FUNCTION_BLOCK MECH2_MDL (* Motion/Fault Model of a Bidirectional Linear Mechanism (Externally Clocked) *)
  (* Standard: 61499-1; Classification: Model; ApplicationDomain: Simulation; Function: Bidirectional Motion *)
  (* Version 0.0, 2004-09-25, JHC, Rockwell Automation, Derived from MECH2_MDL. *)
  (* Compiler header: package fb.rt.mva; import fb.rt.math.*; *)
  (* Compiler Java IBM Jikes 1.06 *)
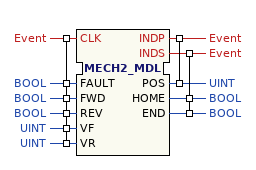
  EVENT_INPUT
    CLK WITH FAULT, FWD, REV, VF, VR; (* External Clock Event *)
  END_EVENT
  EVENT_OUTPUT
    INDP WITH POS; (* Position Changed *)
    INDS WITH HOME, END; (* Sensor Changed *)
  END_EVENT
  VAR_INPUT
    FAULT : BOOL; (* 0=Enable,1=Simulate Fault *)
    FWD : BOOL; (* Move Forward at VF *)
    REV : BOOL; (* Move Back at VR *)
    VF : UINT; (* Forward speed in % Full Scale per CLK event *)
    VR : UINT; (* Reverse speed in %FS per CLK event *)
  END_VAR
  VAR_OUTPUT
    POS : UINT; (* Position,{0..100}percent *)
    HOME : BOOL := 1; (* HOME position limit switch with hysteresis *)
    END : BOOL; (* END position limit switch with hysteresis *)
  END_VAR
  ALGORITHM CLK IN Java:
if(FAULT.value) return;
int speed = FWD.value? VF.value : 0;
if(REV.value) speed -= VR.value;
if(speed==0) return;
if(END.value&&(speed>0)) return;
if(HOME.value&&(speed<0)) return;
POS.value = Math.max(0,Math.min(100,POS.value+speed));
INDP.serviceEvent(this);
boolean oldhome = HOME.value;
boolean oldend = END.value;
HOME.value = (POS.value==0);
END.value = (POS.value==100);
if((HOME.value!=oldhome)||(END.value != oldend)) INDS.serviceEvent(this);
  END_ALGORITHM
END_FUNCTION_BLOCK
